SUBAPPLICATION Uebung_079a_AUI (* COGSOG Speed Over Ground auf UT ausgeben mit AR_Timeout_Zero (Adapter Version) *)
  (* Standard: 61499-2; Description: Copyright (c) 2026 Meisterschulen am Ostbahnhof This program and the accompanying materials are made available under the terms of the Eclipse Public License 2.0 which is available at https://www.eclipse.org/legal/epl-2.0/ SPDX-License-Identifier: EPL-2.0 *)
  (* Version 1.0, 2026-09-17, Franz Höpfinger, Meisterschulen am Ostbahnhof, COGSOG Speed over Ground (Rapid Update) mit PHYS Skalierung (0.036) und AR_Timeout_Zero Fendt-Schaltung (Adapter Version, analog Krauternter TECU_COGSOG.SUB) *)
  PACKAGE Uebungen;
  IMPORT Uebungen::const::UT::TECU::DefaultPool_TECU_Numeric::NumberVariable_Ground_based_machine_speed_N;
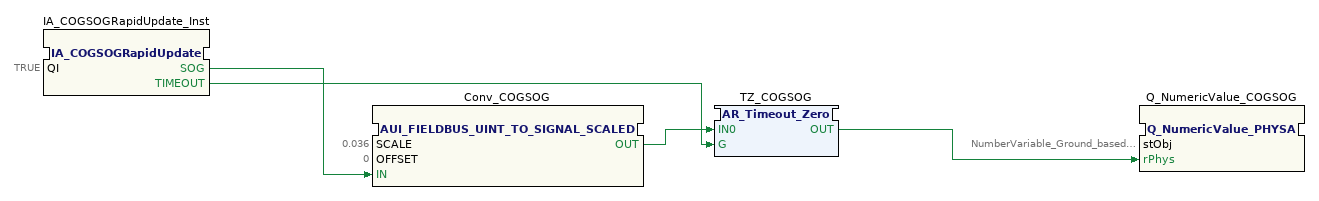
  FBS
    IA_COGSOGRapidUpdate_Inst : isobus::tecu::IA_COGSOGRapidUpdate(QI := TRUE);
    Conv_COGSOG : logiBUS::signalprocessing::fieldbus::AUI_FIELDBUS_UINT_TO_SIGNAL_SCALED(SCALE := 0.036, OFFSET := 0);
    Q_NumericValue_COGSOG : isobus::UT::Q::Q_NumericValue_PHYSA(stObj := NumberVariable_Ground_based_machine_speed_N);
  END_FBS
  SUBAPPS
    TZ_COGSOG : MyLib::sys::AR_Timeout_Zero;
  END_SUBAPPS
  ADAPTER_CONNECTIONS
    IA_COGSOGRapidUpdate_Inst.SOG TO Conv_COGSOG.IN;
    Conv_COGSOG.OUT TO TZ_COGSOG.IN0;
    IA_COGSOGRapidUpdate_Inst.TIMEOUT TO TZ_COGSOG.G;
    TZ_COGSOG.OUT TO Q_NumericValue_COGSOG.rPhys;
  END_CONNECTIONS
END_SUBAPPLICATION
